FUNCTION_BLOCK RT_E_MERGE (* Merge(OR)of multiple events *)
  (* Description: Copyright (c) 2008 ACIN This program and the accompanying materials are made available under the terms of the Eclipse Public License 2.0 which is available at https://www.eclipse.org/legal/epl-2.0/ SPDX-License-Identifier: EPL-2.0 *)
  (* Version 1.0, 2008-07-10, Alois Zoitl, ACIN *)
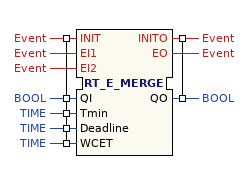
  EVENT_INPUT
    INIT WITH QI, Tmin, Deadline, WCET;
    EI1; (* First input event *)
    EI2; (* Second input event *)
  END_EVENT
  EVENT_OUTPUT
    INITO WITH QO;
    EO; (* Output Event *)
  END_EVENT
  VAR_INPUT
    QI : BOOL;
    Tmin : TIME;
    Deadline : TIME;
    WCET : TIME;
  END_VAR
  VAR_OUTPUT
    QO : BOOL;
  END_VAR
END_FUNCTION_BLOCK
